# EPICS autosave request: iocBoot/common.req
$(P):$(N):ENABLE
$(P):$(N):INT.INPB
$(P):$(N):INT.INPC
